// TIA Portal V20 export
TYPE "HMI_MotSpdCL"
   STRUCT
      FwdMan : Bool;   // 1=Start: Forward Start Command in Manual Mode
      StopMan : Bool;   // 1=Stop: Stop Command in Manual Mode
      RevMan : Bool;   // 1=Start: Reverse Start Command in Manual Mode
      DvFdOnMan : Bool;   // 1=On: Device feed-in On Command in Manual Mode
      DvFdOffMan : Bool;   // 1=Off: Device feed-in Off Command in Manual Mode
      AutModOp : Bool;   // 1=Auto Mode: Auto Mode by Operator
      ManModOp : Bool := TRUE;   // 1=Manual Mode: Manual Mode by Operator
      LocalLi : Bool;   // 1=Local Mode: Local Operation by Field Signal
      LocalOp : Bool;   // 1=Local Mode: Local Operation by Operator
      OosOp : Bool;   // 1=Oos Mode: Oos Mode by Operator
      FwdLocal : Bool;   // 1=Start Local: Field Forward Start Signal
      StopLocal : Bool;   // 1=Stop Local: Field Stop Signal
      RevLocal : Bool;   // 1=Start Local: Field Reverse Start Signal
      SP_Int : Real := 1.0;   // Setpoint (Internal)
      SP_Ext : Real;   // Setpoint (External)
      SP_HiLim : Real := 100.0;   // Setpoint High Limit
      SP_LoLim : Real;   // Setpoint Low Limit
      SP_ExtOp : Bool;   // Operator Input to Select External Setpoint
      SP_IntOp : Bool := TRUE;   // Operator Input to Select Internal Setpoint
      SP_TrkExt : Bool;   // Bumpless Transfer from External to Internal
      SP_RateOn : Bool;   // 1= Activate limitation of setpoint gradients
      SP_RmpOn : Bool;   // 1= Activate setpoint ramp to target SP_RmpTarget
      SP_RmpModTime : Bool;   // 1= Use time SP_RmpTime for ramp, 0= Use rates SP_UpRaLim, SP_DnRaLim
      SP_UpRaLim : Real := 100.0;   // Upward rate limit for setpoint
      SP_DnRaLim : Real := 100.0;   // Downward rate limit for setpoint
      SP_RmpTime : Real;   // Setpoint ramp time [s,min,h]
      SP_RmpTarget : Real;   // Setpoint ramp target
      SP_OpScale : "ScaVal";   // SP - Bar Display Limits for OS
      SP_Unit : Int;   // Engineering units of SP
      RbkUnit : Int;   // Engineering units of Rbk
      RbkWH_Lim : Real := 90.0;   // Rbk - High Warning Limit
      RbkWL_Lim : Real := 10.0;   // Rbk - Low Warning Limit
      RbkHyst : Real := 1.0;   // Rbk - Hysteresis
      RbkOpScale : "ScaVal";   // Rbk - Bar Display Limits for OS
      ER_AH_Lim : Real := 100.0;   // ER alarm high limit
      ER_AL_Lim : Real := -100.0;   // ER alarm low limit
      ER_Hyst : Real := 1.0;   // Hysteresis for ER alarms
      ER_AH_DFac : Real;   // ER alarm coming delay factor for positive SP jump [s/PV_Unit]
      ER_AL_DFac : Real;   // ER alarm coming delay factor for negative SP jump [s/PV_Unit]
      Monitor : Bool := TRUE;   // 1=Monitor ON, 0=Monitor OFF: Feedback Monitor
      MonTiStatic : Real := 3.0;   // Monitoring Time of Feedback [s]
      MonTiDynamic : Real := 3.0;   // Monitoring Time of Feedback on starting or on change in control output [s]
      MonTiDyStop : Real := 3.0;   // Monitoring Time of Feedback on stopping in control output [s]
      RapidStp : Bool;   // 1 = Motor Rapid Stop command
      RstOp : Bool;   // Operator Reset Signal
      Permit_ST : Byte := BYTE#16#FF;   // Permit Signal Status
      Intlock_ST : Byte := BYTE#16#FF;   // Intlock Signal Status
      Protect_ST : Byte := BYTE#16#FF;   // Protect Signal Status
      TimeFactor : Int;   // Time Conversion Factor (0- Sec, 1- Min, 2- Hour)
      CurrMon { ExternalWritable := 'False'} : DInt;   // Remaining monitoring time [s]
      FbkFwdOut { ExternalWritable := 'False'} : Bool;   // 1=Run, 0=Stop: Feedback of Control Forward
      FbkRevOut { ExternalWritable := 'False'} : Bool;   // 1=Run, 0=Stop: Feedback of Control Reverse
      SP_Out { ExternalWritable := 'False'} : Real;   // Analog Output Value
      SP_RateTarget { ExternalWritable := 'False'} : Real;   // Target for limitation of setpoint gradients
      SP_RemRT { ExternalWritable := 'False'} : Real;   // Remaining ramp time of setpoint
      RbkOut { ExternalWritable := 'False'} : Real;   // Readback value output
      OS_PermOut { ExternalWritable := 'False'} : DWord := DWORD#16#FFFF_FFFF;   // Operator Permission: Output for OS
      OS_PermLog { ExternalWritable := 'False'} : DWord := DWORD#16#FFFF_FFFF;   // Operator Permission: Output for OS
      OS1PermOut { ExternalWritable := 'False'} : DWord := DWORD#16#FFFF_FFFF;   // Operator Permission: Output for OS
      OS1PermLog { ExternalWritable := 'False'} : DWord := DWORD#16#FFFF_FFFF;   // Operator Permission: Output for OS
      OpSt_Out { ExternalWritable := 'False'} : DWord;   // Enabled operator stations
      ST_Worst { ExternalWritable := 'False'} : Byte := 16#80;   // Worst Signal Status
      AutoST { ExternalWritable := 'False'} : Byte := 16#80;   // Worst Signal Status of the automatic commands
      Status1 { ExternalWritable := 'False'} : DWord;   // Status1 Word
      Status2 { ExternalWritable := 'False'} : DWord;   // Status2 Word
      Status3 { ExternalWritable := 'False'} : DWord;   // Status3 Word
      Status4 { ExternalWritable := 'False'} : DWord;   // Status4 Word
      Status5 { ExternalWritable := 'False'} : DWord;   // Status5 Word
      AlarmState { ExternalWritable := 'False'} : Word;   // Alarm State for group display / Alarm Status for group display
   END_STRUCT;
   // // SP_OpScale.High : High Value
   // // SP_OpScale.Low : Low Value
   // // RbkOpScale.High : High Value
   // // RbkOpScale.Low : Low Value
END_TYPE
